(* CODESYS project GIT_Binary.project
   Project Profile: RtuProfile

Project tree, tasks and I/O mapping:
  Device : HX3040, Altus S.A., order no. HX3040, version 1.0.0.158
      settings: Primary CPU = 'B2103A42-FB24-495D-AB96-83E194CED7A8'
    application Application
      libraries: LibPlcStandard, 1.0.0.6 (Manufacturer); LibRtuStandard, 1.0.0.11 (Manufacturer); LibDataTypes, 1.0.0.0 (Manufacturer); HX3040 Diagnostic Structs, 1.0.0.3 (Manufacturer); HX8300 Diagnostic Structs, 1.0.0.0 (Manufacturer); NX1001 Diagnostic Structs, 1.0.0.4 (WAA); NX1005 Diagnostic Structs, 1.0.0.4 (WAA); NX2001 Diagnostic Structs, 1.0.0.5 (WAA); NX2020 Diagnostic Structs, 1.0.0.4 (WAA); NX4000 Diagnostic Structs, 1.0.0.0 (WAA); NX6000 Diagnostic Structs, 0.0.0.2 (WAA); NX6100 Diagnostic Structs, 0.0.0.2 (WAA); NX6010 Diagnostic Structs, 0.0.0.5 (Manufacturer); NX6014 Diagnostic Structs, 1.0.0.0 (Manufacturer); NX6020 Diagnostic Structs, 1.0.0.3 (Manufacturer); HX1100 Diagnostic Structs, 0.0.0.2 (Manufacturer); HX1120 Diagnostic Structs, 1.0.0.1 (Manufacturer); HX2200 Diagnostic Structs, 0.0.0.3 (Manufacturer); HX2300 Diagnostic Structs, 0.0.0.1 (Manufacturer); HX2320 Diagnostic Structs, 1.0.0.0 (Manufacturer); HX6000 Diagnostic Structs, 1.0.0.0 (Manufacturer); HX6020 Diagnostic Structs, 1.0.0.0 (Manufacturer); HX6065 Diagnostic Structs, 1.0.0.2 (Manufacturer); NJ1001 Diagnostic Structs, 1.0.0.0 (Manufacturer); NJ1005 Diagnostic Structs, 1.0.0.1 (Manufacturer); NJ2001 Diagnostic Structs, 1.0.0.0 (Manufacturer); NJ6000 Diagnostic Structs, 1.0.0.1 (Manufacturer); NJ6001 Diagnostic Structs, 1.0.0.3 (Manufacturer); NJ6005 Diagnostic Structs, 1.0.0.9 (Manufacturer); NJ6010 Diagnostic Structs, 1.0.0.0 (Manufacturer); NJ6011 Diagnostic Structs, 1.0.0.0 (Manufacturer); NJ6020 Diagnostic Structs, 1.0.0.3 (Manufacturer); NJ6100 Diagnostic Structs, 1.0.0.0 (Manufacturer); NJ6101 Diagnostic Structs, 1.0.0.1 (Manufacturer); Standard, 3.5.12.0 (System)
      task MainTask (cyclic, interval 20 ms, priority 13, watchdog 1000 ms x 1) calls MainPrg
      Diagnostic Explorer
      Bill of Materials
      Configuration and Consumption
      SystemGVLs/
        global variables System_Diagnostics
        global variables Module_Diagnostics
        global variables IOQualities
      UserGVLs/
        global variables Qualities
        global variables ReqDiagnostics
        global variables Disables
      SystemPOUs/
        program MainPrg [ST]
        program EngineeringPrg [ST]
        program AlarmPrg [ST]
      UserPOUs/
        program UserPrg [ST]
        program StartPrg [ST]
    Configuration : Bus, Altus S.A., order no. Configuration, version 1.1.1.1
        settings: Machine Profile = True
      HX3040 : HX3040, Altus S.A., order no. HX3040, version 1.0.0.158
          settings: DC sync0 cycletime = 4000; Rack Configuration Info.Total Number of Racks = 1; Rack Configuration Info.Rack-0 Type = 19001; IOModule's Address for interrupt = 255; Size of the rack where CPU is = 9; CurrentProjectProfileParameter = 'RtuProfile'
        <Vazio>
        COM 1
        COM 2
        NET 1
            settings: IP Address = [192, 168, 200, 96]; Gateway Address = [192, 168, 200, 253]; Obtain Ip automatic = False
        NET 2
        NET 3
        NET 4
        NET 5
        NET 6
        HX8300 : HX8300, Altus S.A., order no. HX8300, version 0.0.0.5
            settings: Physical Address of the Slave = 31; DC sync0 cycletime = 4000; Diag Instance Id = 31
            unmapped channels: %IB0 Digital Inputs - Byte 0
*)

// Device/Application/SystemGVLs/System_Diagnostics
VAR_GLOBAL
	//DG_HX3040 diagnostics variable
	DG_HX3040 : T_DIAG_HX3040_1;
END_VAR

// Device/Application/SystemGVLs/Module_Diagnostics
VAR_GLOBAL
	//DG_HX8300 diagnostics variable
	DG_HX8300 : T_DIAG_HX8300_1;
END_VAR

// Device/Application/UserGVLs/Qualities
VAR_GLOBAL
END_VAR

// Device/Application/UserGVLs/ReqDiagnostics
VAR_GLOBAL
END_VAR

// Device/Application/UserGVLs/Disables
VAR_GLOBAL
END_VAR

// Device/Application/SystemGVLs/IOQualities
VAR_GLOBAL
END_VAR

// Device/Application/SystemPOUs/MainPrg
(*Main POU associated with MainTask that calls StartPrg, UserPrg, NonSkippedPrg and the system POUs AlarmPrg and EngineeringPrg. This POU is blocked to edit.*)
PROGRAM MainPrg
VAR
   isFirstCycle : BOOL := TRUE;
END_VAR

IF isFirstCycle THEN
   StartPrg();
   isFirstCycle := FALSE;
ELSE
   EngineeringPrg();
   AlarmPrg();
   UserPrg();
END_IF;

END_PROGRAM

// Device/Application/UserPOUs/StartPrg
(*The code inserted by the user into this POU is executed once after startup. Before this fist cycle it is not executed again. In case of redundant system, this one is executed in both CPUs during the startup.*)
PROGRAM StartPrg
VAR
END_VAR

END_PROGRAM

// Device/Application/SystemPOUs/EngineeringPrg
(*This POU is blocked to edit and it is generated automatically according the Engineering Screen configurations.*)
PROGRAM EngineeringPrg
VAR
END_VAR

END_PROGRAM

// Device/Application/SystemPOUs/AlarmPrg
(*This POU is blocked to edit and it is generated automatically according the Alarm Screen configurations.*)
PROGRAM AlarmPrg
VAR
END_VAR

END_PROGRAM

// Device/Application/UserPOUs/UserPrg
(*The main code inserted by the user and executed associated with the MainTask must be inserted into this POU.*)
PROGRAM UserPrg
VAR
END_VAR

END_PROGRAM
